INTERFACE IShelfElement EXTENDS __System.IQueryInterface

PROPERTY isOccupied : BOOL
GET
END_GET
SET
END_SET
END_PROPERTY

PROPERTY part : IPart
GET
END_GET
SET
END_SET
END_PROPERTY

END_INTERFACE

(* stored: Version 1.1.0.1
   Itf IShelfElement: Id {e7e6a03c-e907-449d-820d-42f4fa64c398}
   Property isOccupied: Id {547b9917-fc67-4bfb-ae0e-9272d2a52196}
   Get Get: Id {33273cc6-5bfa-4954-8eda-7e21e31f4a3a}
   Set Set: Id {0d3febe8-7e58-4dfc-9b31-0a1a489fbee5}
   Property part: Id {8637dcc2-0164-485b-8793-1704ef10be62}
   Get Get: Id {7e3041fa-e039-4378-b6a2-a537eed22e9b}
   Set Set: Id {84692091-b236-4b41-abc2-f93af9faad09} *)
